{attribute 'hide_all_locals'}
FUNCTION_BLOCK ROTAXIS_BECKHOFF EXTENDS FB_2_ROB_AXIS
VAR_INPUT
	NCAxis : AXIS_REF;
    SETTINGS : stSettings_Axis := (
        MinPosition := -3.141592653589793,
        MaxPosition := 3.141592653589793,
        PositionTolerance := 0.001,
        AngularStandStillLimit := 0.001,
        SafePositionTolerance := 0.001,
        StandardUnits := (
            Position := eUnit.mm,
            Orientation := eUnit.rad,
            Joint := eUnit.rad,
            LinearVelocity := eUnit.mm,
            AngularVelocity := eUnit.rad,
            JointVelocity := eUnit.rad,
            LinearAcceleration := eUnit.mm,
            AngularAcceleration := eUnit.rad,
            JointAcceleration := eUnit.rad));
END_VAR
VAR_IN_OUT
    
END_VAR
VAR_OUTPUT
    AXIS_COMM : FB_3_COMM_AXIS_BECKHOFF;
END_VAR

AXIS_COMM(
        Axis := NCAxis,
        StopVelocityTolerance := SETTINGS.AngularStandStillLimit);
COMM := ADR(AXIS_COMM);
SET_A := SETTINGS;

Powered := AXIS_COMM.Powered;
Homed := AXIS_COMM.Homed;
ActualAxisPosition := AXIS_COMM.ActualPosition;
ActualAxisVelocity := AXIS_COMM.ActualVelocity;

TCPPos_PLCUnit := SETTINGS.InstallationPose;
TCPPos_PLCUnit.yaw := TCPPos_PLCUnit.yaw + _axisActualPosition;
TCPVel_PLCUnit.x := 0.0;
TCPVel_PLCUnit.y := 0.0;
TCPVel_PLCUnit.z := 0.0;
TCPVel_PLCUnit.roll := 0.0;
TCPVel_PLCUnit.pitch := 0.0;
TCPVel_PLCUnit.yaw := _axisActualVelocity;
CYCLIC_AXIS();

METHOD CommandHandler : UINT
VAR_INPUT
    Cmd : eCommands;
    Settings : stCommand_Settings;
END_VAR
VAR
    NewCommandID : UINT;
    TargetPosition : LREAL;
    TargetValid : BOOL;
    EffectiveVelocity : LREAL;
    EffectiveAcceleration : LREAL;
    Accepted : BOOL;
END_VAR
CommandHandler := 0;
IF NOT PrepareAxisCommand(
    Cmd := Cmd,
    Settings := Settings,
    NewCommandID => NewCommandID,
    TargetPosition => TargetPosition,
    TargetValid => TargetValid,
    EffectiveVelocity => EffectiveVelocity,
    EffectiveAcceleration => EffectiveAcceleration) THEN RETURN; END_IF

CASE Cmd OF
    eCommands.MoveL, eCommands.MoveJ, eCommands.MoveJJoints:
        Accepted := AXIS_COMM.SendMoveAbsolute(
            CommandID := NewCommandID,
            Position := TargetPosition,
            Velocity := EffectiveVelocity,
            Acceleration := EffectiveAcceleration,
            Deceleration := SET_A.DefaultDeceleration,
            Jerk := SET_A.DefaultJerk);
    eCommands.MoveLRelativ, eCommands.MoveJRelativ:
        Accepted := AXIS_COMM.SendMoveRelative(
            CommandID := NewCommandID,
            Distance := Settings.Pose.x,
            Velocity := EffectiveVelocity,
            Acceleration := EffectiveAcceleration,
            Deceleration := SET_A.DefaultDeceleration,
            Jerk := SET_A.DefaultJerk);
    eCommands.Homing:
        Accepted := AXIS_COMM.SendHome(CommandID := NewCommandID);
END_CASE

IF Accepted THEN
    CommandHandler := CommitAxisCommand(
        NewCommandID := NewCommandID,
        TargetPosition := TargetPosition,
        TargetValid := TargetValid);
END_IF
END_METHOD

METHOD PROTECTED OnActivate : eResult
VAR
    eParentResult : eResult;
    myResult : eResult;
END_VAR


eParentResult := SUPER^.OnActivate();
myResult := eResult.NONE;

IF eParentResult <> eResult.SUCCESS THEN
    OnActivate := eParentResult;
    RETURN;
END_IF

AXIS_COMM.Power(Enable := FALSE);
IF NOT AXIS_COMM.Powered THEN
    myResult := eResult.SUCCESS;
END_IF

OnActivate := CombineResults(eParentResult, myResult);
END_METHOD

METHOD PROTECTED OnConfigure : eResult
VAR
    eParentResult : eResult;
    myResult : eResult;
END_VAR


eParentResult := SUPER^.OnConfigure();

IF NOT ValidateConfiguration() THEN
    myResult := eResult.FAILURE;
ELSE
    myResult := eResult.SUCCESS;
END_IF

OnConfigure := CombineResults(eParentResult, myResult);
END_METHOD

METHOD PROTECTED OnDeactivate : eResult
VAR
    eParentResult : eResult;
    myResult : eResult;
END_VAR
eParentResult := SUPER^.OnDeactivate();
myResult := eResult.NONE;

IF (ABS(AXIS_COMM.ActualVelocity) > SETTINGS.AngularStandStillLimit) OR AXIS_COMM.Busy THEN
    AXIS_COMM.StopMotion();
ELSE
    AXIS_COMM.Power(Enable := FALSE);
    IF NOT AXIS_COMM.Powered THEN
        myResult := eResult.SUCCESS;
    END_IF
END_IF

OnDeactivate := CombineResults(eParentResult, myResult);
END_METHOD

METHOD PROTECTED OnError : eResult
VAR
    eParentResult : eResult;
    myResult : eResult;
END_VAR
eParentResult := SUPER^.OnError();
myResult := eResult.NONE;

IF eParentResult <> eResult.SUCCESS THEN
    OnError := eParentResult;
    RETURN;
END_IF

IF AXIS_COMM.MESSENGER.HasActivError THEN
    AXIS_COMM.ResetAxis();
    myResult := eResult.NONE;
ELSE
    myResult := eResult.SUCCESS;
END_IF

OnError := CombineResults(eParentResult, myResult);
END_METHOD

END_FUNCTION_BLOCK

(* stored: Version 1.1.0.1, ProductVersion 3.1.4026.18
   POU ROTAXIS_BECKHOFF: Id {317064f0-d9b0-43a6-b27e-f453e25a795f}, SpecialFunc None
   Folder StateControl: Id {9b35bad9-5bf5-4f5d-9198-346680c4ff69}
   Method CommandHandler: Id {ea381757-862d-4cb8-a0c2-e5e461d335e1}
   Method OnActivate: Id {e6d3f096-20dd-424e-bfa4-d0e3f153a517}
   Method OnConfigure: Id {7c207b89-8675-42c1-93c8-982126ff1ee5}
   Method OnDeactivate: Id {8c896843-75b1-4d44-85df-347250d34322}
   Method OnError: Id {921aacc9-c817-44dd-ad83-5c9389c91d41} *)
